// TIA Portal V18 export
// export: Created 2026-06-23T08:49:30.6756926Z, ExportSetting WithDefaults, DisplayName Totally Integrated Automation Portal, DisplayVersion V18, DisplayName TIA Portal Openness, DisplayVersion V18, DisplayName TIA Portal Version Control Interface, DisplayVersion V18, DisplayName STEP 7 Professional, DisplayVersion V18, DisplayName STEP 7 Safety, DisplayVersion V18, DisplayName WinCC Professional, DisplayVersion V18
FUNCTION "FC_VFD_Bon2_Hybrid" : Void   // FC70, LAD
{ S7_Optimized_Access := 'TRUE' }
VERSION : 0.1
// stored: AutoNumber true, IsIECCheckEnabled false, SetENOAutomatically false, UDAEnableTagReadback false
BEGIN

REGION Network 1: Điều khiển contactor VFD Bồn 2
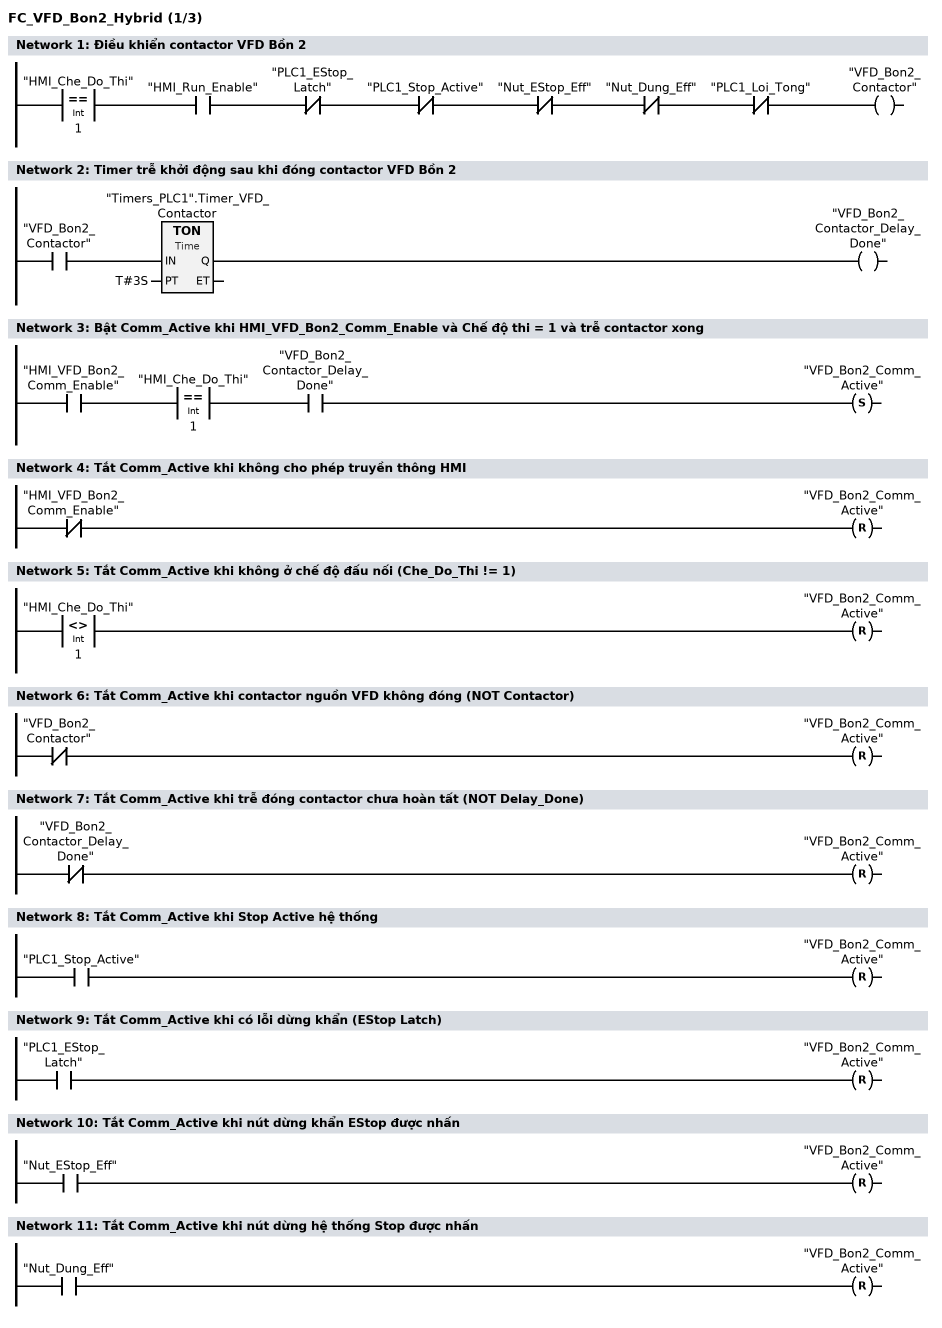
   RUNG wire#powerrail
      { S7_Templates := "SrcType := Int" } EQ_Contact(in1 := "HMI_Che_Do_Thi", in2 := 1)
      Contact( "HMI_Run_Enable" )
      I_Contact( "PLC1_EStop_Latch" )
      I_Contact( "PLC1_Stop_Active" )
      I_Contact( "Nut_EStop_Eff" )
      I_Contact( "Nut_Dung_Eff" )
      I_Contact( "PLC1_Loi_Tong" )
      Coil( "VFD_Bon2_Contactor" )
   END_RUNG
   // the same network as SCL:
   "VFD_Bon2_Contactor" := ("HMI_Che_Do_Thi" = 1) AND "HMI_Run_Enable" AND NOT "PLC1_EStop_Latch" AND NOT "PLC1_Stop_Active" AND NOT "Nut_EStop_Eff" AND NOT "Nut_Dung_Eff" AND NOT "PLC1_Loi_Tong";
END_REGION

REGION Network 2: Timer trễ khởi động sau khi đóng contactor VFD Bồn 2
   RUNG wire#powerrail
      Contact( "VFD_Bon2_Contactor" )
      { S7_Templates := "time_type := Time" } "Timers_PLC1".Timer_VFD_Contactor.TON(pt := T#3S, et =>)
      Coil( "VFD_Bon2_Contactor_Delay_Done" )
   END_RUNG
   // the same network as SCL:
   "Timers_PLC1".Timer_VFD_Contactor.TON(IN := "VFD_Bon2_Contactor", PT := T#3S);
   "VFD_Bon2_Contactor_Delay_Done" := "Timers_PLC1".Timer_VFD_Contactor.Q;
END_REGION

REGION Network 3: Bật Comm_Active khi HMI_VFD_Bon2_Comm_Enable và Chế độ thi = 1 và trễ contactor xong
   RUNG wire#powerrail
      Contact( "HMI_VFD_Bon2_Comm_Enable" )
      { S7_Templates := "SrcType := Int" } EQ_Contact(in1 := "HMI_Che_Do_Thi", in2 := 1)
      Contact( "VFD_Bon2_Contactor_Delay_Done" )
      S_Coil( "VFD_Bon2_Comm_Active" )
   END_RUNG
   // the same network as SCL:
   IF "HMI_VFD_Bon2_Comm_Enable" AND ("HMI_Che_Do_Thi" = 1) AND "VFD_Bon2_Contactor_Delay_Done" THEN
       "VFD_Bon2_Comm_Active" := TRUE;
   END_IF;
END_REGION

REGION Network 4: Tắt Comm_Active khi không cho phép truyền thông HMI
   RUNG wire#powerrail
      I_Contact( "HMI_VFD_Bon2_Comm_Enable" )
      R_Coil( "VFD_Bon2_Comm_Active" )
   END_RUNG
   // the same network as SCL:
   IF NOT "HMI_VFD_Bon2_Comm_Enable" THEN "VFD_Bon2_Comm_Active" := FALSE; END_IF;
END_REGION

REGION Network 5: Tắt Comm_Active khi không ở chế độ đấu nối (Che_Do_Thi != 1)
   RUNG wire#powerrail
      { S7_Templates := "SrcType := Int" } NE_Contact(in1 := "HMI_Che_Do_Thi", in2 := 1)
      R_Coil( "VFD_Bon2_Comm_Active" )
   END_RUNG
   // the same network as SCL:
   IF "HMI_Che_Do_Thi" <> 1 THEN "VFD_Bon2_Comm_Active" := FALSE; END_IF;
END_REGION

REGION Network 6: Tắt Comm_Active khi contactor nguồn VFD không đóng (NOT Contactor)
   RUNG wire#powerrail
      I_Contact( "VFD_Bon2_Contactor" )
      R_Coil( "VFD_Bon2_Comm_Active" )
   END_RUNG
   // the same network as SCL:
   IF NOT "VFD_Bon2_Contactor" THEN "VFD_Bon2_Comm_Active" := FALSE; END_IF;
END_REGION

REGION Network 7: Tắt Comm_Active khi trễ đóng contactor chưa hoàn tất (NOT Delay_Done)
   RUNG wire#powerrail
      I_Contact( "VFD_Bon2_Contactor_Delay_Done" )
      R_Coil( "VFD_Bon2_Comm_Active" )
   END_RUNG
   // the same network as SCL:
   IF NOT "VFD_Bon2_Contactor_Delay_Done" THEN "VFD_Bon2_Comm_Active" := FALSE; END_IF;
END_REGION

REGION Network 8: Tắt Comm_Active khi Stop Active hệ thống
   RUNG wire#powerrail
      Contact( "PLC1_Stop_Active" )
      R_Coil( "VFD_Bon2_Comm_Active" )
   END_RUNG
   // the same network as SCL:
   IF "PLC1_Stop_Active" THEN "VFD_Bon2_Comm_Active" := FALSE; END_IF;
END_REGION

REGION Network 9: Tắt Comm_Active khi có lỗi dừng khẩn (EStop Latch)
   RUNG wire#powerrail
      Contact( "PLC1_EStop_Latch" )
      R_Coil( "VFD_Bon2_Comm_Active" )
   END_RUNG
   // the same network as SCL:
   IF "PLC1_EStop_Latch" THEN "VFD_Bon2_Comm_Active" := FALSE; END_IF;
END_REGION

REGION Network 10: Tắt Comm_Active khi nút dừng khẩn EStop được nhấn
   RUNG wire#powerrail
      Contact( "Nut_EStop_Eff" )
      R_Coil( "VFD_Bon2_Comm_Active" )
   END_RUNG
   // the same network as SCL:
   IF "Nut_EStop_Eff" THEN "VFD_Bon2_Comm_Active" := FALSE; END_IF;
END_REGION

REGION Network 11: Tắt Comm_Active khi nút dừng hệ thống Stop được nhấn
   RUNG wire#powerrail
      Contact( "Nut_Dung_Eff" )
      R_Coil( "VFD_Bon2_Comm_Active" )
   END_RUNG
   // the same network as SCL:
   IF "Nut_Dung_Eff" THEN "VFD_Bon2_Comm_Active" := FALSE; END_IF;
END_REGION

REGION Network 12: Tắt Comm_Active khi hệ thống báo lỗi tổng (Loi_Tong)
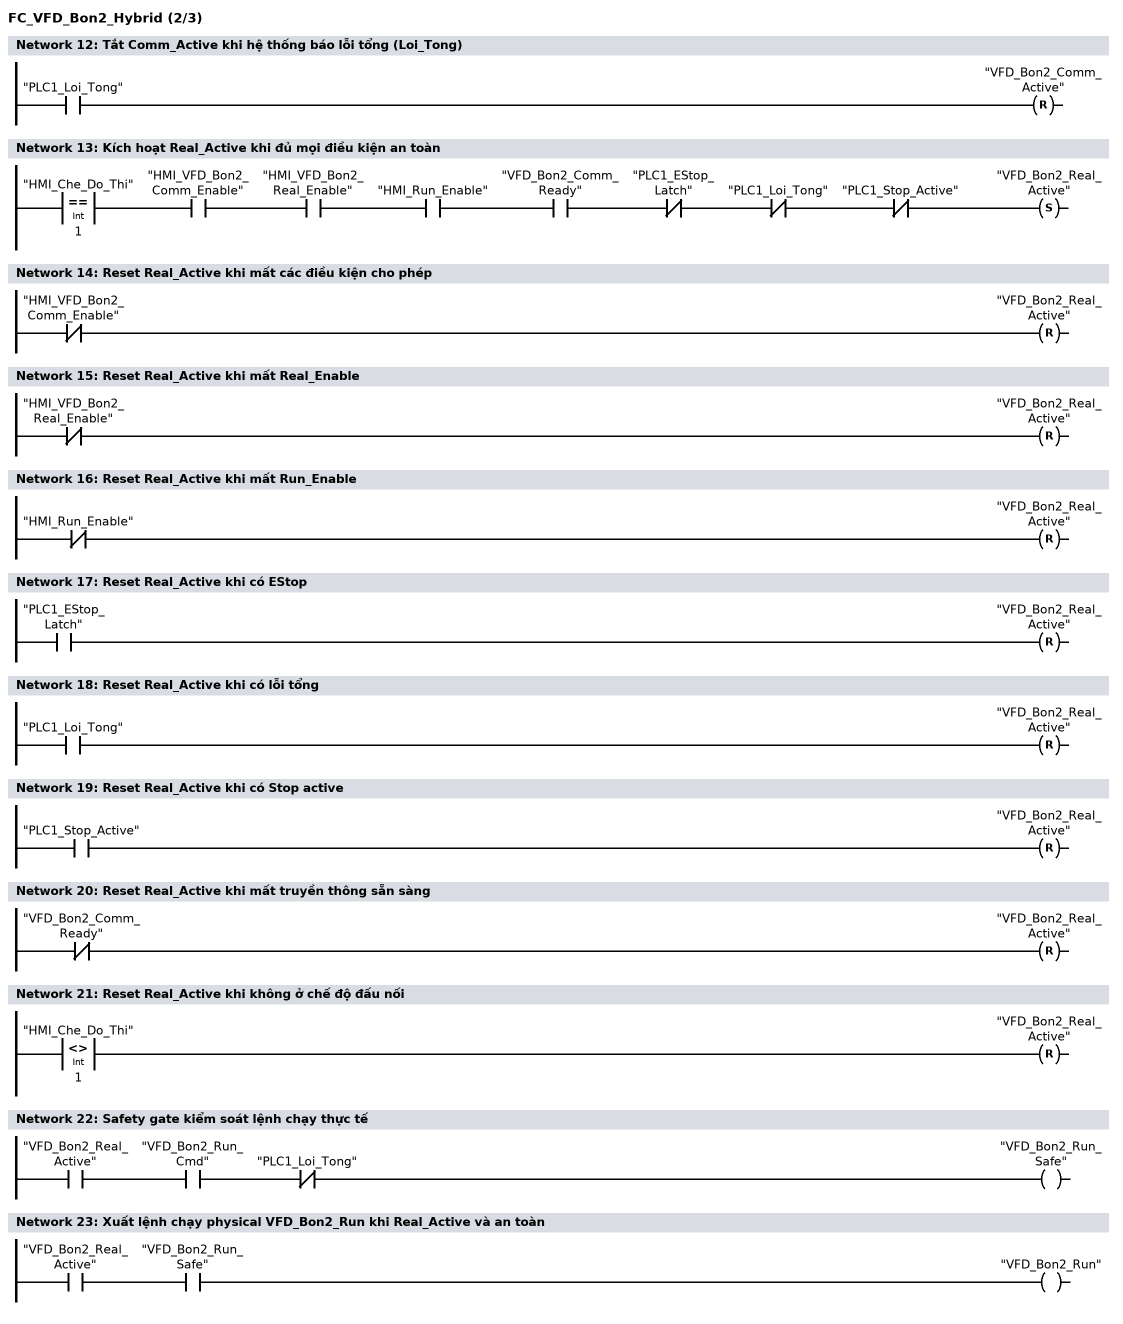
   RUNG wire#powerrail
      Contact( "PLC1_Loi_Tong" )
      R_Coil( "VFD_Bon2_Comm_Active" )
   END_RUNG
   // the same network as SCL:
   IF "PLC1_Loi_Tong" THEN "VFD_Bon2_Comm_Active" := FALSE; END_IF;
END_REGION

REGION Network 13: Kích hoạt Real_Active khi đủ mọi điều kiện an toàn
   RUNG wire#powerrail
      { S7_Templates := "SrcType := Int" } EQ_Contact(in1 := "HMI_Che_Do_Thi", in2 := 1)
      Contact( "HMI_VFD_Bon2_Comm_Enable" )
      Contact( "HMI_VFD_Bon2_Real_Enable" )
      Contact( "HMI_Run_Enable" )
      Contact( "VFD_Bon2_Comm_Ready" )
      I_Contact( "PLC1_EStop_Latch" )
      I_Contact( "PLC1_Loi_Tong" )
      I_Contact( "PLC1_Stop_Active" )
      S_Coil( "VFD_Bon2_Real_Active" )
   END_RUNG
   // the same network as SCL:
   IF ("HMI_Che_Do_Thi" = 1) AND "HMI_VFD_Bon2_Comm_Enable" AND "HMI_VFD_Bon2_Real_Enable" AND "HMI_Run_Enable" AND "VFD_Bon2_Comm_Ready" AND NOT "PLC1_EStop_Latch" AND NOT "PLC1_Loi_Tong" AND NOT "PLC1_Stop_Active" THEN
       "VFD_Bon2_Real_Active" := TRUE;
   END_IF;
END_REGION

REGION Network 14: Reset Real_Active khi mất các điều kiện cho phép
   RUNG wire#powerrail
      I_Contact( "HMI_VFD_Bon2_Comm_Enable" )
      R_Coil( "VFD_Bon2_Real_Active" )
   END_RUNG
   // the same network as SCL:
   IF NOT "HMI_VFD_Bon2_Comm_Enable" THEN "VFD_Bon2_Real_Active" := FALSE; END_IF;
END_REGION

REGION Network 15: Reset Real_Active khi mất Real_Enable
   RUNG wire#powerrail
      I_Contact( "HMI_VFD_Bon2_Real_Enable" )
      R_Coil( "VFD_Bon2_Real_Active" )
   END_RUNG
   // the same network as SCL:
   IF NOT "HMI_VFD_Bon2_Real_Enable" THEN "VFD_Bon2_Real_Active" := FALSE; END_IF;
END_REGION

REGION Network 16: Reset Real_Active khi mất Run_Enable
   RUNG wire#powerrail
      I_Contact( "HMI_Run_Enable" )
      R_Coil( "VFD_Bon2_Real_Active" )
   END_RUNG
   // the same network as SCL:
   IF NOT "HMI_Run_Enable" THEN "VFD_Bon2_Real_Active" := FALSE; END_IF;
END_REGION

REGION Network 17: Reset Real_Active khi có EStop
   RUNG wire#powerrail
      Contact( "PLC1_EStop_Latch" )
      R_Coil( "VFD_Bon2_Real_Active" )
   END_RUNG
   // the same network as SCL:
   IF "PLC1_EStop_Latch" THEN "VFD_Bon2_Real_Active" := FALSE; END_IF;
END_REGION

REGION Network 18: Reset Real_Active khi có lỗi tổng
   RUNG wire#powerrail
      Contact( "PLC1_Loi_Tong" )
      R_Coil( "VFD_Bon2_Real_Active" )
   END_RUNG
   // the same network as SCL:
   IF "PLC1_Loi_Tong" THEN "VFD_Bon2_Real_Active" := FALSE; END_IF;
END_REGION

REGION Network 19: Reset Real_Active khi có Stop active
   RUNG wire#powerrail
      Contact( "PLC1_Stop_Active" )
      R_Coil( "VFD_Bon2_Real_Active" )
   END_RUNG
   // the same network as SCL:
   IF "PLC1_Stop_Active" THEN "VFD_Bon2_Real_Active" := FALSE; END_IF;
END_REGION

REGION Network 20: Reset Real_Active khi mất truyền thông sẵn sàng
   RUNG wire#powerrail
      I_Contact( "VFD_Bon2_Comm_Ready" )
      R_Coil( "VFD_Bon2_Real_Active" )
   END_RUNG
   // the same network as SCL:
   IF NOT "VFD_Bon2_Comm_Ready" THEN "VFD_Bon2_Real_Active" := FALSE; END_IF;
END_REGION

REGION Network 21: Reset Real_Active khi không ở chế độ đấu nối
   RUNG wire#powerrail
      { S7_Templates := "SrcType := Int" } NE_Contact(in1 := "HMI_Che_Do_Thi", in2 := 1)
      R_Coil( "VFD_Bon2_Real_Active" )
   END_RUNG
   // the same network as SCL:
   IF "HMI_Che_Do_Thi" <> 1 THEN "VFD_Bon2_Real_Active" := FALSE; END_IF;
END_REGION

REGION Network 22: Safety gate kiểm soát lệnh chạy thực tế
   RUNG wire#powerrail
      Contact( "VFD_Bon2_Real_Active" )
      Contact( "VFD_Bon2_Run_Cmd" )
      I_Contact( "PLC1_Loi_Tong" )
      Coil( "VFD_Bon2_Run_Safe" )
   END_RUNG
   // the same network as SCL:
   "VFD_Bon2_Run_Safe" := "VFD_Bon2_Real_Active" AND "VFD_Bon2_Run_Cmd" AND NOT "PLC1_Loi_Tong";
END_REGION

REGION Network 23: Xuất lệnh chạy physical VFD_Bon2_Run khi Real_Active và an toàn
   RUNG wire#powerrail
      Contact( "VFD_Bon2_Real_Active" )
      Contact( "VFD_Bon2_Run_Safe" )
      Coil( "VFD_Bon2_Run" )
   END_RUNG
   // the same network as SCL:
   "VFD_Bon2_Run" := "VFD_Bon2_Real_Active" AND "VFD_Bon2_Run_Safe";
END_REGION

REGION Network 24: Xuất lệnh đảo chiều physical VFD_Bon2_Dao_Chieu khi Real_Active
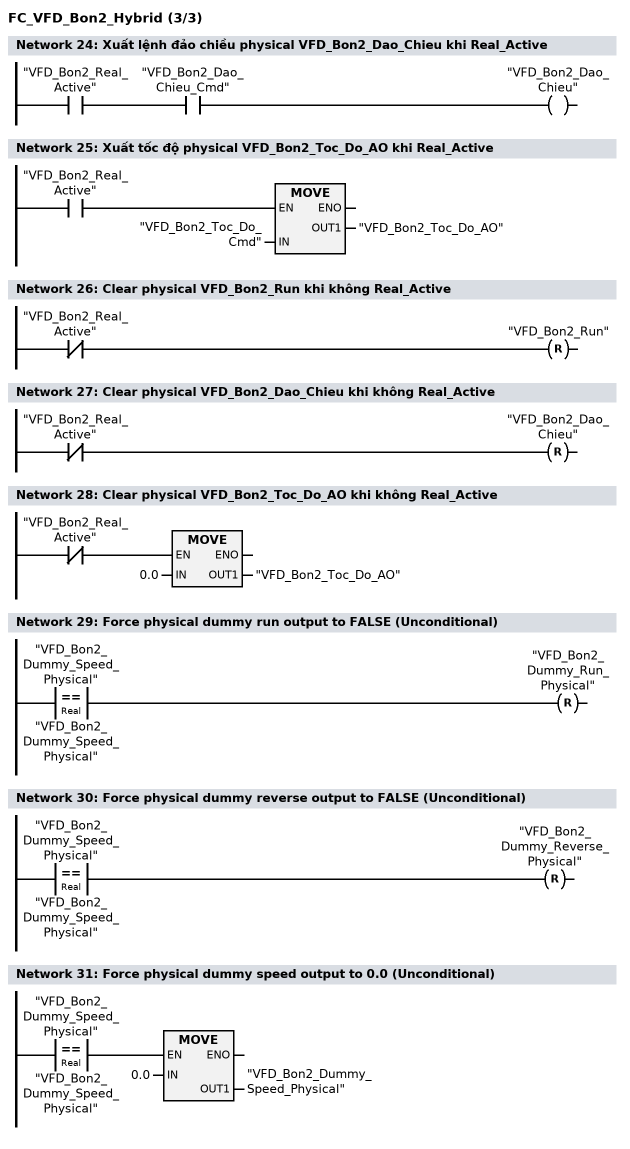
   RUNG wire#powerrail
      Contact( "VFD_Bon2_Real_Active" )
      Contact( "VFD_Bon2_Dao_Chieu_Cmd" )
      Coil( "VFD_Bon2_Dao_Chieu" )
   END_RUNG
   // the same network as SCL:
   "VFD_Bon2_Dao_Chieu" := "VFD_Bon2_Real_Active" AND "VFD_Bon2_Dao_Chieu_Cmd";
END_REGION

REGION Network 25: Xuất tốc độ physical VFD_Bon2_Toc_Do_AO khi Real_Active
   RUNG wire#powerrail
      Contact( "VFD_Bon2_Real_Active" )
      { S7_GenerateENO := "TRUE" } Move(in := "VFD_Bon2_Toc_Do_Cmd", out1 => "VFD_Bon2_Toc_Do_AO")
   END_RUNG
   // the same network as SCL:
   IF "VFD_Bon2_Real_Active" THEN "VFD_Bon2_Toc_Do_AO" := "VFD_Bon2_Toc_Do_Cmd"; END_IF;
END_REGION

REGION Network 26: Clear physical VFD_Bon2_Run khi không Real_Active
   RUNG wire#powerrail
      I_Contact( "VFD_Bon2_Real_Active" )
      R_Coil( "VFD_Bon2_Run" )
   END_RUNG
   // the same network as SCL:
   IF NOT "VFD_Bon2_Real_Active" THEN "VFD_Bon2_Run" := FALSE; END_IF;
END_REGION

REGION Network 27: Clear physical VFD_Bon2_Dao_Chieu khi không Real_Active
   RUNG wire#powerrail
      I_Contact( "VFD_Bon2_Real_Active" )
      R_Coil( "VFD_Bon2_Dao_Chieu" )
   END_RUNG
   // the same network as SCL:
   IF NOT "VFD_Bon2_Real_Active" THEN "VFD_Bon2_Dao_Chieu" := FALSE; END_IF;
END_REGION

REGION Network 28: Clear physical VFD_Bon2_Toc_Do_AO khi không Real_Active
   RUNG wire#powerrail
      I_Contact( "VFD_Bon2_Real_Active" )
      { S7_GenerateENO := "TRUE" } Move(in := 0.0, out1 => "VFD_Bon2_Toc_Do_AO")
   END_RUNG
   // the same network as SCL:
   IF NOT "VFD_Bon2_Real_Active" THEN "VFD_Bon2_Toc_Do_AO" := 0.0; END_IF;
END_REGION

REGION Network 29: Force physical dummy run output to FALSE (Unconditional)
   RUNG wire#powerrail
      { S7_Templates := "SrcType := Real" } EQ_Contact(in1 := "VFD_Bon2_Dummy_Speed_Physical", in2 := "VFD_Bon2_Dummy_Speed_Physical")
      R_Coil( "VFD_Bon2_Dummy_Run_Physical" )
   END_RUNG
   // the same network as SCL:
   IF "VFD_Bon2_Dummy_Speed_Physical" = "VFD_Bon2_Dummy_Speed_Physical" THEN
       "VFD_Bon2_Dummy_Run_Physical" := FALSE;
   END_IF;
END_REGION

REGION Network 30: Force physical dummy reverse output to FALSE (Unconditional)
   RUNG wire#powerrail
      { S7_Templates := "SrcType := Real" } EQ_Contact(in1 := "VFD_Bon2_Dummy_Speed_Physical", in2 := "VFD_Bon2_Dummy_Speed_Physical")
      R_Coil( "VFD_Bon2_Dummy_Reverse_Physical" )
   END_RUNG
   // the same network as SCL:
   IF "VFD_Bon2_Dummy_Speed_Physical" = "VFD_Bon2_Dummy_Speed_Physical" THEN
       "VFD_Bon2_Dummy_Reverse_Physical" := FALSE;
   END_IF;
END_REGION

REGION Network 31: Force physical dummy speed output to 0.0 (Unconditional)
   RUNG wire#powerrail
      { S7_Templates := "SrcType := Real" } EQ_Contact(in1 := "VFD_Bon2_Dummy_Speed_Physical", in2 := "VFD_Bon2_Dummy_Speed_Physical")
      { S7_GenerateENO := "TRUE" } Move(in := 0.0, out1 => "VFD_Bon2_Dummy_Speed_Physical")
   END_RUNG
   // the same network as SCL:
   IF "VFD_Bon2_Dummy_Speed_Physical" = "VFD_Bon2_Dummy_Speed_Physical" THEN
       "VFD_Bon2_Dummy_Speed_Physical" := 0.0;
   END_IF;
END_REGION
END_FUNCTION
